FUNCTION_BLOCK AI_FIELDBUS_INT_TO_SIGNAL (* Mirrors IN->OUT if Signal Valid. *)
  (* Standard: 61499-1 *)
  (* Version 1.0, 2026-05-31, franz *)
  PACKAGE logiBUS::signalprocessing::fieldbus;
  IMPORT signalprocessing::FIELDBUS_SIGNAL::NOT_AVAILABLE_WM;
  IMPORT signalprocessing::FIELDBUS_SIGNAL::VALID_SIGNAL_W;
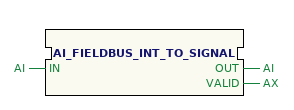
  SOCKETS
    IN : adapter::types::unidirectional::AI; (* Input *)
  END_SOCKETS
  PLUGS
    OUT : adapter::types::unidirectional::AI; (* Output Filtered *)
    VALID : adapter::types::unidirectional::AX; (* TRUE if Signal is VALID *)
  END_PLUGS
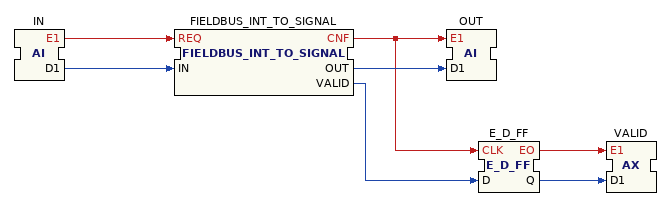
  FBS
    FIELDBUS_INT_TO_SIGNAL : logiBUS::signalprocessing::fieldbus::FIELDBUS_INT_TO_SIGNAL;
    E_D_FF : iec61499::events::E_D_FF;
  END_FBS
  EVENT_CONNECTIONS
    IN.E1 TO FIELDBUS_INT_TO_SIGNAL.REQ;
    FIELDBUS_INT_TO_SIGNAL.CNF TO OUT.E1;
    FIELDBUS_INT_TO_SIGNAL.CNF TO E_D_FF.CLK;
    E_D_FF.EO TO VALID.E1;
  END_CONNECTIONS
  DATA_CONNECTIONS
    IN.D1 TO FIELDBUS_INT_TO_SIGNAL.IN;
    FIELDBUS_INT_TO_SIGNAL.OUT TO OUT.D1;
    FIELDBUS_INT_TO_SIGNAL.VALID TO E_D_FF.D;
    E_D_FF.Q TO VALID.D1;
  END_CONNECTIONS
END_FUNCTION_BLOCK
